// TIA Portal V18 export
ORGANIZATION_BLOCK "Main"   // OB1, LAD, ProgramCycle
TITLE = "Main Program Sweep (Cycle)"
{ S7_Optimized_Access := 'TRUE' }
// stored: SetENOAutomatically false
   VAR_INPUT
      Initial_Call : Bool;   // Initial call of this OB
      Remanence : Bool;   // =True, if remanent data are available
   END_VAR
BEGIN

REGION Network 1
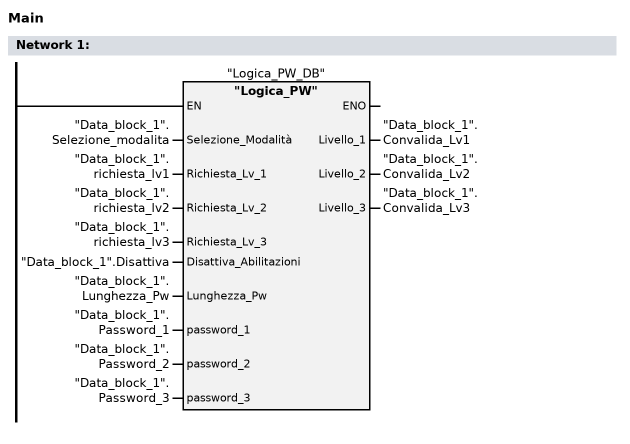
   RUNG wire#powerrail
      "Logica_PW_DB"(Selezione_Modalità := "Data_block_1".Selezione_modalita, Richiesta_Lv_1 := "Data_block_1".richiesta_lv1, Richiesta_Lv_2 := "Data_block_1".richiesta_lv2, Richiesta_Lv_3 := "Data_block_1".richiesta_lv3, Disattiva_Abilitazioni := "Data_block_1".Disattiva, Lunghezza_Pw := "Data_block_1".Lunghezza_Pw, password_1 := "Data_block_1".Password_1, password_2 := "Data_block_1".Password_2, password_3 := "Data_block_1".Password_3, Livello_1 => "Data_block_1".Convalida_Lv1, Livello_2 => "Data_block_1".Convalida_Lv2, Livello_3 => "Data_block_1".Convalida_Lv3)
   END_RUNG
   // the same network as SCL:
   "Logica_PW_DB"(Selezione_Modalità := "Data_block_1".Selezione_modalita,   // "Logica_PW"
                  Richiesta_Lv_1 := "Data_block_1".richiesta_lv1,
                  Richiesta_Lv_2 := "Data_block_1".richiesta_lv2,
                  Richiesta_Lv_3 := "Data_block_1".richiesta_lv3,
                  Disattiva_Abilitazioni := "Data_block_1".Disattiva,
                  Lunghezza_Pw := "Data_block_1".Lunghezza_Pw,
                  password_1 := "Data_block_1".Password_1,
                  password_2 := "Data_block_1".Password_2,
                  password_3 := "Data_block_1".Password_3,
                  Livello_1 => "Data_block_1".Convalida_Lv1,
                  Livello_2 => "Data_block_1".Convalida_Lv2,
                  Livello_3 => "Data_block_1".Convalida_Lv3);
END_REGION
END_ORGANIZATION_BLOCK
